FUNCTION_BLOCK CabinControl (* Basic Function Block Type *)
  (* Standard: 61499-2 *)
  (* Version 0.0, 6/17/2016, Andrei, nxtControl GmbH, Template *)
  PACKAGE Main;
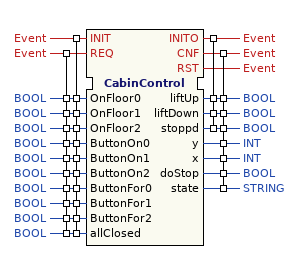
  EVENT_INPUT
    INIT WITH OnFloor0, OnFloor1, OnFloor2, ButtonOn0, ButtonOn1, ButtonOn2, ButtonFor0, ButtonFor1, ButtonFor2, allClosed; (* Initialization Request *)
    REQ WITH OnFloor0, OnFloor1, OnFloor2, ButtonOn0, ButtonOn1, ButtonOn2, ButtonFor0, ButtonFor1, ButtonFor2, allClosed; (* Normal Execution Request *)
  END_EVENT
  EVENT_OUTPUT
    INITO WITH liftUp, liftDown, stoppd; (* Initialization Confirm *)
    CNF WITH liftUp, liftDown, stoppd, y, x, doStop, state; (* Execution Confirmation *)
    RST;
  END_EVENT
  VAR_INPUT
    OnFloor0 : BOOL; (* Input event qualifier *)
    OnFloor1 : BOOL;
    OnFloor2 : BOOL;
    ButtonOn0 : BOOL;
    ButtonOn1 : BOOL;
    ButtonOn2 : BOOL;
    ButtonFor0 : BOOL;
    ButtonFor1 : BOOL;
    ButtonFor2 : BOOL;
    allClosed : BOOL;
  END_VAR
  VAR_OUTPUT
    liftUp : BOOL;
    liftDown : BOOL; (* Output event qualifier *)
    stoppd : BOOL;
    y : INT;
    x : INT;
    doStop : BOOL;
    state : STRING;
  END_VAR
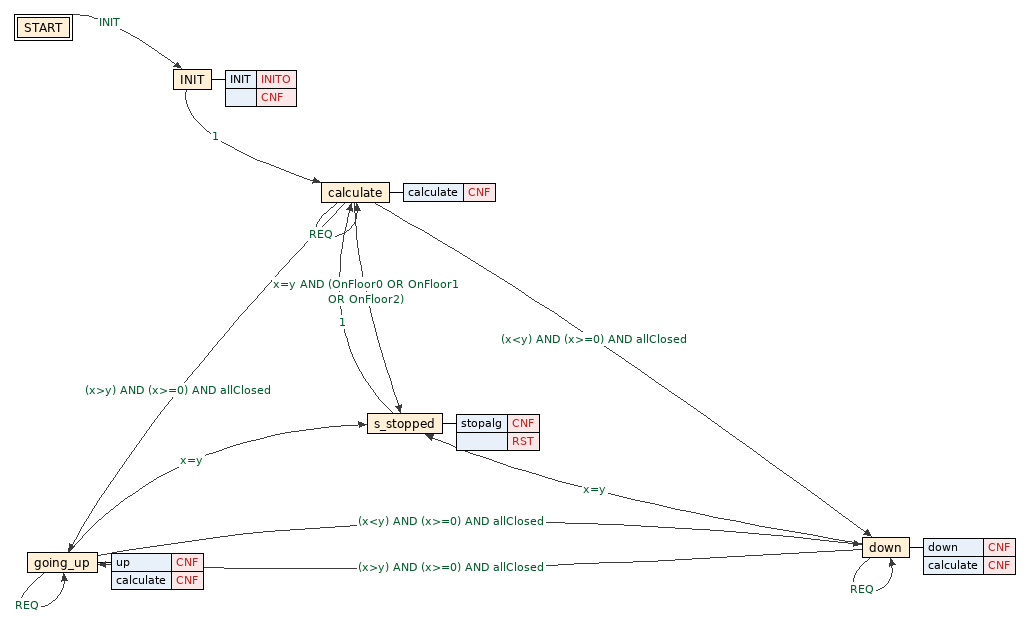
  EC_STATES
    START; (* Initial State *)
    INIT : INIT -> INITO, -> CNF;
    going_up : up -> CNF, calculate -> CNF;
    s_stopped : stopalg -> CNF, -> RST;
    down : down -> CNF, calculate -> CNF;
    calculate : calculate -> CNF;
  END_STATES
  EC_TRANSITIONS
    START TO INIT := INIT;
    calculate TO going_up := (x>y) AND (x>=0)  AND allClosed;
    INIT TO calculate := 1;
    calculate TO down := (x<y) AND (x>=0) AND allClosed;
    down TO s_stopped := x=y;
    calculate TO calculate := REQ;
    down TO down := REQ;
    going_up TO going_up := REQ;
    down TO going_up := (x>y) AND (x>=0)  AND allClosed;
    going_up TO s_stopped := x=y;
    going_up TO down := (x<y) AND (x>=0) AND allClosed;
    s_stopped TO calculate := 1;
    calculate TO s_stopped := x=y AND (OnFloor0 OR OnFloor1 OR OnFloor2);
  END_TRANSITIONS
  ALGORITHM stopalg IN ST:
;
state := 'STOP';
liftUp := FALSE;
liftDown := FALSE;
stoppd := TRUE;
  END_ALGORITHM
  ALGORITHM up IN ST:
;
state := 'UP';
liftUp := TRUE;
liftDown := FALSE;
stoppd := FALSE;
(* To continue going if all OnFloor are false*)
IF NOT OnFloor0 OR NOT OnFloor1 OR NOT OnFloor2 THEN
	y := 3;
END_IF;
  END_ALGORITHM
  ALGORITHM down IN ST:
;
state := 'DOWN';
liftUp := FALSE;
liftDown := TRUE;
stoppd := FALSE;
(* To continue going if all OnFloor are false*)
IF NOT OnFloor0 OR NOT OnFloor1 OR NOT OnFloor2 THEN
	y := -1;
END_IF;
  END_ALGORITHM
  ALGORITHM calculate IN ST:
(* Determine the current floor *)
IF ButtonOn0 OR ButtonFor0 THEN
	x:=0;
ELSIF ButtonOn1 OR ButtonFor1 THEN
	x:=1;
ELSIF ButtonOn2 OR ButtonFor2 THEN
	x:=2;
END_IF;

IF OnFloor0 THEN
	y:=0;
ELSIF OnFloor1 THEN
	y:=1;
ELSIF OnFloor2 THEN
	y:=2;
END_IF;
  END_ALGORITHM
  ALGORITHM INIT IN ST:
;
y := 2;
x :=2;
  END_ALGORITHM
END_FUNCTION_BLOCK
